// TIA Portal V19 export
TYPE "LEXCHANGETRAY_typeConstraintWorkstationEm_toConstraintRollerFeedback"
// stored: Access Published
   STRUCT
      transferEnable : Bool;   // 请求转移
      unConstrainting : Bool;   // 解拘束中
      unConstrainted : Bool;   // 解拘束完成
   END_STRUCT;
END_TYPE
